FUNCTION_BLOCK "FB_ProductionLineControl"
{ S7_Optimized_Access := 'TRUE' }

   VAR_INPUT
      Mode : BOOL; // 用于切换生产线的手动和自动模式
      ForwardButton : BOOL; // 正转按钮
      ReverseButton : BOOL; // 反转按钮
      SensorA : BOOL; // 传感器A
      SensorB : BOOL; // 传感器B
      SensorC : BOOL; // 传感器C
      ButtonA : BOOL; // 按钮A
      ButtonB : BOOL; // 按钮B
      ButtonC : BOOL; // 按钮C
   END_VAR

   VAR_OUTPUT
      MotorForward : BOOL; // 电机正转输出
      MotorReverse : BOOL; // 电机反转输出
      CompletionLight : BOOL; // 产品加工完成指示灯
   END_VAR

   VAR
      State : INT; // 状态机当前状态
   END_VAR


BEGIN
   // 状态机初始化
   IF #State = 0 THEN
      #MotorForward := FALSE;
      #MotorReverse := FALSE;
      #CompletionLight := FALSE;
      #State := 1; // 初始状态
   END_IF;

   // 手动模式
   IF #Mode = FALSE THEN
      IF #ForwardButton AND NOT #ReverseButton THEN
         #MotorForward := TRUE;
         #MotorReverse := FALSE;
      ELSIF #ReverseButton AND NOT #ForwardButton THEN
         #MotorReverse := TRUE;
         #MotorForward := FALSE;
      ELSE
         #MotorForward := FALSE;
         #MotorReverse := FALSE;
      END_IF;
   ELSE // 自动模式
      CASE #State OF
         1: // 等待产品到达A
            IF #SensorA THEN
               #State := 2;
            END_IF;
         2: // 等待按钮A按下
            IF #ButtonA THEN
               #MotorForward := TRUE;
               #State := 3;
            END_IF;
         3: // 等待产品到达B
            IF #SensorB THEN
               #MotorForward := FALSE;
               #State := 4;
            END_IF;
         4: // 等待按钮B按下
            IF #ButtonB THEN
               #MotorForward := TRUE;
               #State := 5;
            END_IF;
         5: // 等待产品到达C
            IF #SensorC THEN
               #MotorForward := FALSE;
               #State := 6;
            END_IF;
         6: // 等待按钮C按下
            IF #ButtonC THEN
               #CompletionLight := TRUE;
               #State := 7;
            END_IF;
         7: // 等待产品被取走
            IF NOT #SensorC THEN
               #CompletionLight := FALSE;
               #State := 1;
            END_IF;
      END_CASE;
   END_IF;
END_FUNCTION_BLOCK
